// TIA Portal V16 export
// export: Created 2026-06-17T17:02:33.8698928Z, ExportSetting WithDefaults, DisplayName Totally Integrated Automation Portal, DisplayVersion V16 Update 8, DisplayName TIA Portal Version Control Interface, DisplayVersion V16 Update 8, DisplayName TIA Portal Openness, DisplayVersion V16 Update 8, DisplayName SINAMICS Startdrive Advanced, DisplayVersion V16, DisplayName SINAMICS Startdrive G130, G150, S120, S150, SINAMICS MV, S210, DisplayVersion V16, DisplayName SINAMICS Startdrive G110M, G120, G120C, G120D, G120P, DisplayVersion V16, DisplayName STEP 7 Professional, DisplayVersion V16 Update 8, DisplayName STEP 7 Safety, DisplayVersion V16 Update 7, DisplayName WinCC Advanced, DisplayVersion V16 Update 8
Screen "Motor_Control"  1280x800, Number=1
  ScreenLayer "Motor_Control"
    IOField "I/O 域_1" at 270,166 size 1280x800  DataFormat=Decimal, FormatPattern=9999999, Mode=InOutput
    Button "按钮_1" at 406,60 size 1280x800  Mode=Text, TextOff="Text", TextOn="Text"
    SymbolicIOField "符号 I/O 域_1" at 177,87 size 1280x800  CountVisibleItems=3, Mode=InOutput, OnValue=1, TextOff="0", TextOn="1"
    Circle "圆_1" at 457,199 size 1280x800
    TextField "文本域_1" at 140,178 size 1280x800  Text="Text"
